TYPE ST_CalibrationReportHeader :
STRUCT
	sReportId          : STRING(50);
    sCalibrationNo     : STRING(30);
    sUserId            : STRING(50);
    sDensity           : STRING(30);
    sSolventNo         : STRING(30);
    sSolventRevision   : STRING(30);
    sSysRevisionNo     : STRING(30);
    sAllowableFail     : STRING(30);
    sReplicates        : STRING(30);
    sCallInterval      : STRING(30);
    sCreatedAt         : STRING(30);
END_STRUCT
END_TYPE

(* stored: Version 1.1.0.1, ProductVersion 3.1.4024.15
   DUT ST_CalibrationReportHeader: Id {cc848bc9-fdb0-4d30-aa77-b46d8a2b4145} *)
